FUNCTION_BLOCK FB_CTManagerDefGrid EXTENDS FB_CTManager
VAR_INPUT
END_VAR
VAR_OUTPUT
END_VAR
VAR
  fbContainerInstances    : ARRAY[0..lC_MAX_CTS-1] OF FB_ContainerDefGrid;   // NOTE: 0 based array like base in library
END_VAR

// call CT manager base
SUPER^();

// call specific CT implementation
nCtr := 0;
WHILE nCtr < nListCount DO
  nIndx := ((nListTail + nCtr) MOD lC_MAX_CTS);    // calculate element index in list
  
  // cyclic call of CT body
  fbContainerInstances[nIndx]();
  
  nCtr := nCtr + 1;
END_WHILE

updateLogLevels();

(*
  Abort CTs
*)
METHOD AbortCts : BOOL
VAR_INPUT
  iCT : I_CT;     // reference CT 
  nSel : INT;     // selection: -1=all older (created before reference), 0=current only, 1=all newer (created after reference)
  Src : REFERENCE TO T_ErrSrc;
END_VAR
VAR
  iIterCt : I_CT;
  pCtSelected : POINTER TO FB_ContainerDefGrid;
END_VAR

// WARNING: This function is NOT tested!!! 
//    TODO: remove this comments when tested

IF nSel = 0 THEN
  // Abort referenced CT
  pCtSelected := GetContainerInstance(iCT:=iCT);
  IF pCtSelected <> 0 THEN
    pCtSelected^.AbortDeformation(sReason:=F_Concat2('CTM Abort CTs Sel=', TO_STRING(nSel)), Src:=Src, bHideLog:=FALSE);
  END_IF
  
ELSIF nSel < 0 THEN
  // Abort previous
  iIterCt := iCT;
  WHILE iIterCt.pListPrev <> 0 DO
    // get instance and abort
    pCtSelected := GetContainerInstance(iCT:=iIterCt);
    IF pCtSelected <> 0 THEN
      pCtSelected^.AbortDeformation(sReason:=F_Concat2('CTM Abort CTs Sel=', TO_STRING(nSel)), Src:=Src, bHideLog:=FALSE);
    END_IF
    // select prev
    iIterCt := iIterCt.pListPrev;
  END_WHILE
  
ELSIF nSel > 0 THEN  
  // Abort next
  iIterCt := iCT;
  WHILE iIterCt.pListNext <> 0 DO
    // get instance and abort
    pCtSelected := GetContainerInstance(iCT:=iIterCt);
    IF pCtSelected <> 0 THEN
      pCtSelected^.AbortDeformation(sReason:=F_Concat2('CTM Abort CTs Sel=', TO_STRING(nSel)), Src:=Src, bHideLog:=FALSE);
    END_IF
    // select next
    iIterCt := iIterCt.pListNext;
  END_WHILE
END_IF
END_METHOD

(*
  Get specific container reference (pointer) from container interface.
*)
METHOD PUBLIC GetContainerInstance : POINTER TO FB_ContainerDefGrid
VAR_INPUT
  iCT              : I_CT;          (*container at triggered event position*)
END_VAR
VAR
  nCtSel             : UDINT;
END_VAR
IF iCT = 0 THEN LogError(Msg:='GetContainerInstance invalid container'); RETURN; END_IF
nCtSel := iCT.pCT^.nMemIndex;
IF nCtSel < lC_MAX_CTS THEN
  GetContainerInstance := ADR( fbContainerInstances[nCtSel] );
END_IF
END_METHOD

METHOD Init
VAR
  nCtr      : UDINT;
END_VAR
// init FB_CTManager(base) list (interface I_CT) with specific Container instances (FBs) 
FOR nCtr := 0 TO lC_MAX_CTS-1 DO
  iContainerList[nCtr] := fbContainerInstances[nCtr];
END_FOR

// call parent init
SUPER^.InitBase(bAutoDelete:=TRUE);
END_METHOD

PROPERTY sCTDefGridInstancesPath : STRING
GET
// build path tho one image deformation fb
// e.g. PRG_PRINT.fbCTM.fbContainerInstances[%id%].fBImageDeformation where %id% will be resolved later in the pyhton script.
//      array in plc lower bound is index 0
sCTDefGridInstancesPath := F_CONCAT2(THIS^.InstanceName, '.fbContainerInstances[%id%].fBImageDeformation');
END_GET
END_PROPERTY

METHOD PRIVATE updateLogLevels
VAR_INST
  _LogLvl_mem  : E_LogSeverity;
END_VAR
// logLevel update from manager to all containers
IF LogLevel <> _LogLvl_mem THEN 
  nCtr := 0;
  WHILE nCtr < lC_MAX_CTS DO
    fbContainerInstances[nCtr].LogLevel := LogLevel;
    nCtr := nCtr + 1;
  END_WHILE
END_IF

_LogLvl_mem := LogLevel;
END_METHOD

END_FUNCTION_BLOCK

(* stored: Version 1.1.0.1, ProductVersion 3.1.4024.11
   POU FB_CTManagerDefGrid: Id {64e24f37-1762-4987-94b6-1c2daabf0872}, SpecialFunc None
   Method AbortCts: Id {887d2e55-f283-4461-92bd-fe8efb68fdd3}
   Method GetContainerInstance: Id {4019ff74-9ad2-43f1-90de-a88d411277f4}
   Method Init: Id {322a3013-e920-45b4-8f41-4730c09f6a49}
   Property sCTDefGridInstancesPath: Id {b4d88d3c-ac8f-4c1b-9101-ee6ed3ea35b7}
   Get Get: Id {d342d67e-171a-43aa-9516-1ffc59a514cc}
   Method updateLogLevels: Id {c5b2038e-8748-4e32-b316-bccf513e122a} *)
